(* PLC project flour_weighing, Dassault Systèmes ControlBuild 2024x Refresh1 *)
(* stored: creationDateTime 2024-04-12T14:05:57-01:00 *)

FUNCTION_BLOCK copie_batch.flour_weighing
  VAR_INPUT
    weighingRequest : BOOL := false;
    cycleInProgress : BOOL := false;
    weighedWeight : DINT := 0;
  END_VAR
  VAR_INPUT
    flourWeight : DINT := 0;
  END_VAR
  VAR_OUTPUT
    weighingOk : BOOL := false;
  END_VAR
  VAR_OUTPUT
    introduceFlour : BOOL := false;
    introFlourEnd : BOOL := false;
    exitFlour : BOOL := false;
    exitFlourEnd : BOOL := false;
  END_VAR
  VAR
    totalWeight : DINT := 0;
    endOfWeighing : BOOL := false;
  END_VAR
  VAR CONSTANT
    maxWeight : DINT := 100;
  END_VAR

INITIAL_STEP 10:
  10_INLINE1(N);
  COMPUTE_FUNCTION_BLOCKS(S);
END_STEP
ACTION 10_INLINE1:
  totalWeight := 0;
END_ACTION
TRANSITION FROM 10 TO 11
  := cycleInProgress AND weighingRequest;
END_TRANSITION
STEP 11:
  11_INLINE2(N);
END_STEP
ACTION 11_INLINE2:
  introduceFlour;
END_ACTION
TRANSITION FROM 11 TO 12
  := endOfWeighing;
END_TRANSITION
STEP 12:
  12_INLINE3(N);
END_STEP
ACTION 12_INLINE3:
  IF(RE X12) THEN
  	totalWeight := totalWeight + weighedWeight;
  END_IF;
END_ACTION
TRANSITION FROM 12 TO 13
  := cycleInProgress AND T/X12/250ms;
END_TRANSITION
STEP 13:
  13_INLINE4(N);
END_STEP
ACTION 13_INLINE4:
  exitFlour;
END_ACTION
TRANSITION FROM 13 TO 14
  := cycleInProgress AND (weighedWeight <= 1);
END_TRANSITION
STEP 14:
END_STEP
TRANSITION FROM 14 TO 15
  := cycleInProgress AND (totalWeight >= flourWeight);
END_TRANSITION
TRANSITION FROM 14 TO 11
  := cycleInProgress AND (totalWeight < flourWeight);
END_TRANSITION
STEP 15:
  15_INLINE5(N);
END_STEP
ACTION 15_INLINE5:
  weighingOk;
END_ACTION
TRANSITION FROM 15 TO 10
  := NOT weighingRequest;
END_TRANSITION
ACTION COMPUTE_FUNCTION_BLOCKS:  (* blocks drawn on the SFC sheet *)
  G1:
END_ACTION

ACTION PreSFC:
endOfWeighing := ((totalWeight + weighedWeight) >= flourWeight) 
OR (weighedWeight >= maxWeight);
END_ACTION

ACTION PostSFC:
IF NOT cycleInProgress THEN
	introduceFlour := FALSE;
	exitFlour := FALSE;
END_IF;

introFlourEnd := NOT introduceFlour OR NOT cycleInProgress;
exitFlourEnd := NOT exitFlour OR NOT cycleInProgress;
END_ACTION
END_FUNCTION_BLOCK
